# B&R Automation Studio project RTFProj (part 5)

##### test.c
```c
/*********************************************************************************************
* B&R Automation - Perfection in Automation (https://www.br-automation.com)
    ******************************************************************************************
    * Program 	    : Master's Thesis - Soccer Table (Table Football - real game)
    * Author  	    : Roman Parak
    * Created 	    : date ...
	* University    : Brno University of Technology(BUT)
	* Faculty       : Faculty of Mechanical Engineering(FME)
	* Study Program : Applied Computer Science and Control
	* Institute     : Institute of Automation and Computer Science
**********************************************************************************************
* Implementation OF PROGRAM Test(Real_Game/Technology/Test/Program/test.h)
**********************************************************************************************/

/*************************** LIBRARIES *********************************/
#include <bur/plc.h>
#include <bur/plctypes.h>
#include <stdio.h>
#include <math.h>

#include "rp_funcx1.h"
#include "Structures/test_str.h"
#include "Functions/test_fce.h"

#ifdef _DEFAULT_INCLUDES
	#include <AsDefault.h>
#endif

/*************************** DEFINITIONS *******************************/
#define EACH_FORMATION 1;

/************************ LOCAL VARIABLES ******************************/
// struct - MpAlarmX
_LOCAL MpAlarmXListUIConnectType AlarmListUI_ConnectType;
_LOCAL MpAlarmXHistoryUIConnectType AlarmHistoryUI_ConnectType;
// udint
_LOCAL UDINT alarm_device_address;
// bool
_LOCAL BOOL start;
_LOCAL BOOL stop;
// usint
_LOCAL USINT max_numberOfFormation;
_LOCAL USINT i_axisNum;
// lreal
_LOCAL LREAL temp_lin;
_LOCAL LREAL temp_rot;
_LOCAL LREAL define_posRotary;
_LOCAL LREAL angle_ofRotation;
// state machine
_LOCAL rp_MainSteps soccer_step;

/**********************************************************************************************************/
/********************************************** INIT PROGRAM **********************************************/
/**********************************************************************************************************/
void _INIT ProgramInit(void)
{
    /*********************************** Declaration variables **********************************/
    // generally
    max_numberOfFormation = EACH_FORMATION;

    // axis type -> MAPP
    // linear
    gLinkAxes_linear[0] = gk_mappAxisL;
    /*
    gLinkAxes_linear[1] = df_mappAxisL;
    gLinkAxes_linear[2] = md_mappAxisL;
    gLinkAxes_linear[3] = fw_mappAxisL;
    */
    // rotary
    gLinkAxes_rotary[0] = gk_mappAxisR;
   	/*
    gLinkAxes_rotary[1] = df_mappAxisR;
    gLinkAxes_rotary[2] = md_mappAxisR;
    gLinkAxes_rotary[3] = fw_mappAxisR;
    */
    /************************************ Control of AlarmX ************************************/

    // adjustment device name
    alarm_device_address = (UDINT) strcpy(mp_alarmX.deviceName_no1_exp,"EXPORT_HISTORY");
    // MpAlarmX Core
    mp_alarmX.mp_core.MpLink         = &gAlarmXCore;
    mp_alarmX.mp_core.Enable         = 1;
    // MpAlarmX ListUI
    mp_alarmX.mp_listUI.MpLink       = &gAlarmXCore;
    mp_alarmX.mp_listUI.Enable       = 1;
    mp_alarmX.mp_listUI.UIConnect    = &AlarmListUI_ConnectType;
    // MpAlarmX History
    mp_alarmX.mp_history.MpLink      = &gAlarmXHistory;
    mp_alarmX.mp_history.Enable      = 1;
    mp_alarmX.mp_history.DeviceName  = &mp_alarmX.deviceName_no1_exp;
    // MpAlarmX HistoryUI
    mp_alarmX.mp_historyUI.MpLink    = &gAlarmXHistory;
    mp_alarmX.mp_historyUI.Enable    = 1;
    mp_alarmX.mp_historyUI.UIConnect = &AlarmHistoryUI_ConnectType;

    /************************************* Control of Axes **************************************/

    for(i_axisNum = 0; i_axisNum <= max_numberOfFormation - 1; i_axisNum++){
        // initialization ACOPOS variables through function(get_axisParam), that returns two variables type of UDINT
        // into the structure -> axesAcopos(have two parameters : linear, rotary)
        axis_acopos = get_axisParam(i_axisNum);
        // linear -> LinMot
        // linear axis basic
        mp_Axis.mp_axisLinear[i_axisNum].Enable     = 1;
        mp_Axis.mp_axisLinear[i_axisNum].MpLink     = &gLinkAxes_linear[i_axisNum];
        mp_Axis.mp_axisLinear[i_axisNum].Parameters = &mp_Axis.param_axisLinear[i_axisNum];
        mp_Axis.mp_axisLinear[i_axisNum].Axis       = axis_acopos.linear;
		// initialization parameters -> linear
		mp_Axis.param_axisLinear[i_axisNum].Home.Mode 	 		 	     = mpAXIS_HOME_MODE_BLOCK_TORQUE;
		mp_Axis.param_axisLinear[i_axisNum].Home.Position 		  	     = 900;
		mp_Axis.param_axisLinear[i_axisNum].Home.StartVelocity   		 = 350;
		mp_Axis.param_axisLinear[i_axisNum].Home.HomingVelocity  		 = 450;
		mp_Axis.param_axisLinear[i_axisNum].Home.Acceleration    		 = 350;
		mp_Axis.param_axisLinear[i_axisNum].Home.StartDirection  		 = mpAXIS_HOME_DIR_POSITIVE;
		mp_Axis.param_axisLinear[i_axisNum].Home.HomingDirection 		 = mpAXIS_HOME_DIR_NEGATIVE;
		mp_Axis.param_axisLinear[i_axisNum].Home.TorqueLimit	 		 = 0.05;
		mp_Axis.param_axisLinear[i_axisNum].Home.PositionErrorStopLimit	 = 900;
        // linear cyclic set
        mp_Axis.mp_cyclicSetLinear[i_axisNum].Enable     = 1;
        mp_Axis.mp_cyclicSetLinear[i_axisNum].MpLink     = &gLinkAxes_linear[i_axisNum];
        mp_Axis.mp_cyclicSetLinear[i_axisNum].Parameters = &mp_Axis.param_cyclicSetLinear[i_axisNum];
		// config
		mp_Axis.mp_configAxisLinear[i_axisNum].Enable 		 = 1;
		mp_Axis.mp_configAxisLinear[i_axisNum].MpLink 		 = &gLinkAxes_linear[i_axisNum];
		mp_Axis.mp_configAxisLinear[i_axisNum].Configuration = &mp_Axis.param_configAxisLinear[i_axisNum];
        // rotary -> EnDat
        // rotary axis basic
        mp_Axis.mp_axisRotary[i_axisNum].Enable     = 1;
        mp_Axis.mp_axisRotary[i_axisNum].MpLink     = &gLinkAxes_rotary[i_axisNum];
        mp_Axis.mp_axisRotary[i_axisNum].Parameters = &mp_Axis.param_axisRotary[i_axisNum];
        mp_Axis.mp_axisRotary[i_axisNum].Axis       = axis_acopos.rotary;
        // rotary cyclic set
        mp_Axis.mp_cyclicSetRotary[i_axisNum].Enable     = 1;
        mp_Axis.mp_cyclicSetRotary[i_axisNum].MpLink     = &gLinkAxes_rotary[i_axisNum];
        mp_Axis.mp_cyclicSetRotary[i_axisNum].Parameters = &mp_Axis.param_cyclicSetRotary[i_axisNum];
		// config
		mp_Axis.mp_configAxisRotary[i_axisNum].Enable 		 = 1;
		mp_Axis.mp_configAxisRotary[i_axisNum].MpLink 		 = &gLinkAxes_rotary[i_axisNum];
		mp_Axis.mp_configAxisRotary[i_axisNum].Configuration = &mp_Axis.param_configAxisRotary[i_axisNum];
		// temperature - linear
		mp_Axis.param_axisLinear[i_axisNum].CyclicRead.MotorTempMode = mpAXIS_READ_POLLING_1s;
		// temperature - rotary
		mp_Axis.param_axisRotary[i_axisNum].CyclicRead.MotorTempMode = mpAXIS_READ_POLLING_1s;
    }
	// initializatiom temp
	temp_lin = 0;
	temp_rot = 0;
	define_posRotary = 118520697;
	angle_ofRotation = 0;
	// initialization state machine
	soccer_step = STEP_INITIALIZATION;
}

/**********************************************************************************************************/
/********************************************** MAIN PROGRAM **********************************************/
/**********************************************************************************************************/
void _CYCLIC ProgramCyclic(void)
{
	// initializatiom temp
	temp_lin = mp_Axis.mp_axisLinear[0].Info.CyclicRead.MotorTemperature.Value;
	temp_rot = mp_Axis.mp_axisRotary[0].Info.CyclicRead.MotorTemperature.Value;

	switch(soccer_step)
	{
		case STEP_INITIALIZATION:
			{
				if(mp_Axis.mp_axisLinear[0].Active == 1 && mp_Axis.mp_axisRotary[0].Active == 1){
					angle_ofRotation = get_rotationalPostition(mp_Axis.mp_axisRotary[0].Position,define_posRotary);

					if(labs(angle_ofRotation) <= 3600){
						mp_Axis.param_axisRotary[0].Home.Position = angle_ofRotation;
						soccer_step = STEP_INITIALIZATION0;
					}
				}
			}
			break;
		case STEP_INITIALIZATION0:
			{
				if(mp_Axis.mp_axisLinear[0].Error == 1 && mp_Axis.mp_axisRotary[0].Error == 0){
					soccer_step = STEP_ERROR1;
				}else if(mp_Axis.mp_axisLinear[0].StatusID < 0 || mp_Axis.mp_axisRotary[0].StatusID < 0){
					soccer_step = STEP_ERROR2;
				}else {
					if(mp_Axis.mp_axisLinear[0].IsHomed == 1 && mp_Axis.mp_axisRotary[0].IsHomed == 1){
						soccer_step = STEP_RUN7;
					}else{
						soccer_step = STEP_INITIALIZATION1;
					}
				}
			}
			break;
		case STEP_INITIALIZATION1:
			{
				if(start == 1){
					mp_Axis.mp_axisLinear[0].Power = 1;
					mp_Axis.mp_axisRotary[0].Power = 1;

					if(mp_alarmX.mp_core.ActiveAlarms == 1){
						soccer_step = STEP_ERROR1;
					}else if(stop == 1){
						soccer_step = STEP_STOP1;
					}else{
						if(mp_Axis.mp_axisLinear[0].PowerOn == 1 && mp_Axis.mp_axisRotary[0].PowerOn == 1){
							soccer_step = STEP_INITIALIZATION2;
						}
					}
				}
			}
			break;
		case STEP_INITIALIZATION2:
			{
				mp_Axis.mp_axisLinear[0].Update = 1;
				mp_Axis.mp_axisRotary[0].Update = 1;

				if(mp_alarmX.mp_core.ActiveAlarms == 1){
					soccer_step = STEP_ERROR1;
				}else if(stop == 1){
					soccer_step = STEP_STOP1;
				}else{
					if(mp_Axis.mp_axisLinear[0].UpdateDone == 1 && mp_Axis.mp_axisRotary[0].UpdateDone == 1){
						mp_Axis.mp_axisLinear[0].Update = 0;
						mp_Axis.mp_axisRotary[0].Update = 0;
						soccer_step = STEP_INITIALIZATION3;
					}
				}
			}
			break;
		case STEP_INITIALIZATION3:
			{
				mp_Axis.mp_axisRotary[0].Home = 1;

				if(mp_alarmX.mp_core.ActiveAlarms == 1){
					soccer_step = STEP_ERROR1;
				}else if(stop == 1){
					soccer_step = STEP_STOP1;
				}else{
					if(mp_Axis.mp_axisRotary[0].IsHomed == 1){
						mp_Axis.mp_axisRotary[0].Home = 0;
						soccer_step = STEP_INITIALIZATION4;
					}
				}
			}
			break;
		case STEP_INITIALIZATION4:
			{
				mp_Axis.param_cyclicSetRotary[0].Acceleration = 2000;
				mp_Axis.param_cyclicSetRotary[0].Deceleration = 2000;
				mp_Axis.param_cyclicSetRotary[0].PositionModeMaxVelocity = 85000;
				mp_Axis.mp_cyclicSetRotary[0].Velocity 	 = 1000;
				mp_Axis.mp_cyclicSetRotary[0].Position	 = 0;

				mp_Axis.mp_cyclicSetRotary[0].Update = 1;
				if(mp_alarmX.mp_core.ActiveAlarms == 1){
					soccer_step = STEP_ERROR1;
				}else if(stop == 1){
					soccer_step = STEP_STOP1;
				}else{
					if(mp_Axis.mp_cyclicSetRotary[0].UpdateDone == 1){
						mp_Axis.mp_cyclicSetRotary[0].Update = 0;
						if(mp_Axis.mp_cyclicSetRotary[0].CommandBusy == 0 && mp_Axis.mp_cyclicSetRotary[0].CyclicSetActive == 0){
							soccer_step = STEP_INITIALIZATION5;
						}
					}
				}
			}
			break;
		case STEP_INITIALIZATION5:
			{
				mp_Axis.mp_cyclicSetRotary[0].CyclicPosition = 1;
				if(mp_alarmX.mp_core.ActiveAlarms == 1){
					soccer_step = STEP_ERROR1;
				}else if(stop == 1){
					soccer_step = STEP_STOP1;
				}else{
					if(mp_Axis.mp_cyclicSetRotary[0].Info.SlavePosition == 0){
						mp_Axis.mp_cyclicSetRotary[0].CyclicPosition = 0;
						if(mp_Axis.mp_cyclicSetRotary[0].CommandBusy == 0 && mp_Axis.mp_cyclicSetRotary[0].CyclicSetActive == 0){
							soccer_step = STEP_INITIALIZATION6;
						}
					}
				}
			}
			break;
		case STEP_INITIALIZATION6:
			{
				mp_Axis.mp_axisLinear[0].Home = 1;

				if(mp_alarmX.mp_core.ActiveAlarms == 1){
					soccer_step = STEP_ERROR1;
				}else if(stop == 1){
					soccer_step = STEP_STOP1;
				}else{
					if(mp_Axis.mp_axisLinear[0].IsHomed == 1){
						mp_Axis.mp_axisLinear[0].Home = 0;
						soccer_step = STEP_START;
					}
				}
			}
			break;
		case STEP_START:
			{
				mp_Axis.param_cyclicSetLinear[0].Acceleration = 400000;
				mp_Axis.param_cyclicSetLinear[0].Deceleration = 400000;
				mp_Axis.param_cyclicSetLinear[0].PositionModeMaxVelocity = 30000;
				mp_Axis.mp_cyclicSetLinear[0].Velocity = 19000;
				mp_Axis.mp_cyclicSetLinear[0].Position = 0;

				mp_Axis.mp_cyclicSetLinear[0].Update = 1;
				if(mp_alarmX.mp_core.ActiveAlarms == 1){
					soccer_step = STEP_ERROR1;
				}else if(stop == 1){
					soccer_step = STEP_STOP1;
				}else{
					if(mp_Axis.mp_cyclicSetLinear[0].UpdateDone == 1){
						mp_Axis.mp_cyclicSetLinear[0].Update = 0;
						if(mp_Axis.mp_cyclicSetLinear[0].CommandBusy == 0 && mp_Axis.mp_cyclicSetLinear[0].CyclicSetActive == 0){
							soccer_step = STEP_RUN1;
						}
					}
				}
			}
			break;
		case STEP_RUN1:
			{
				mp_Axis.mp_cyclicSetLinear[0].CyclicPosition = 1;
				if(mp_alarmX.mp_core.ActiveAlarms == 1){
					soccer_step = STEP_ERROR1;
				}else if(stop == 1){
					soccer_step = STEP_STOP1;
				}else{
					if(mp_Axis.mp_cyclicSetLinear[0].Info.SlavePosition == 0){
						mp_Axis.mp_cyclicSetLinear[0].CyclicPosition = 0;
						if(mp_Axis.mp_cyclicSetLinear[0].CommandBusy == 0 && mp_Axis.mp_cyclicSetLinear[0].CyclicSetActive == 0){
							soccer_step = STEP_RUN2;
						}
					}
				}
			}
			break;
		case STEP_RUN2:
			{
				mp_Axis.param_cyclicSetRotary[0].Acceleration = 125000;
				mp_Axis.param_cyclicSetRotary[0].Deceleration = 125000;
				mp_Axis.param_cyclicSetRotary[0].PositionModeMaxVelocity = 85000;
				mp_Axis.mp_cyclicSetRotary[0].Velocity 	 = 10000;
				mp_Axis.mp_cyclicSetRotary[0].Position	 = -800;

				mp_Axis.mp_cyclicSetRotary[0].Update = 1;
				if(mp_alarmX.mp_core.ActiveAlarms == 1){
					soccer_step = STEP_ERROR1;
				}else if(stop == 1){
					soccer_step = STEP_STOP1;
				}else{
					if(mp_Axis.mp_cyclicSetRotary[0].UpdateDone == 1){
						mp_Axis.mp_cyclicSetRotary[0].Update = 0;
						if(mp_Axis.mp_cyclicSetRotary[0].CommandBusy == 0 && mp_Axis.mp_cyclicSetRotary[0].CyclicSetActive == 0){
							soccer_step = STEP_RUN3;
						}
					}
				}
			}
			break;
		case STEP_RUN3:
			{
				mp_Axis.mp_cyclicSetRotary[0].CyclicPosition = 1;
				if(mp_alarmX.mp_core.ActiveAlarms == 1){
					soccer_step = STEP_ERROR1;
				}else if(stop == 1){
					soccer_step = STEP_STOP1;
				}else{
					if(mp_Axis.mp_cyclicSetRotary[0].Info.SlavePosition == -800){
						mp_Axis.mp_cyclicSetRotary[0].CyclicPosition = 0;
						if(mp_Axis.mp_cyclicSetRotary[0].CommandBusy == 0 && mp_Axis.mp_cyclicSetRotary[0].CyclicSetActive == 0){
							soccer_step = STEP_RUN4;
						}
					}
				}
			}
			break;
		case STEP_RUN4:
			{
				mp_Axis.param_cyclicSetRotary[0].Acceleration = 125000;
				mp_Axis.param_cyclicSetRotary[0].Deceleration = 125000;
				mp_Axis.param_cyclicSetRotary[0].PositionModeMaxVelocity = 85000;
				mp_Axis.mp_cyclicSetRotary[0].Velocity 	 = 10000;
				mp_Axis.mp_cyclicSetRotary[0].Position	 = 800;

				mp_Axis.mp_cyclicSetRotary[0].Update = 1;
				if(mp_alarmX.mp_core.ActiveAlarms == 1){
					soccer_step = STEP_ERROR1;
				}else if(stop == 1){
					soccer_step = STEP_STOP1;
				}else{
					if(mp_Axis.mp_cyclicSetRotary[0].UpdateDone == 1){
						mp_Axis.mp_cyclicSetRotary[0].Update = 0;
						if(mp_Axis.mp_cyclicSetRotary[0].CommandBusy == 0 && mp_Axis.mp_cyclicSetRotary[0].CyclicSetActive == 0){
							soccer_step = STEP_RUN5;
						}
					}
				}
			}
			break;
		case STEP_RUN5:
			{
				mp_Axis.mp_cyclicSetRotary[0].CyclicPosition = 1;
				if(mp_alarmX.mp_core.ActiveAlarms == 1){
					soccer_step = STEP_ERROR1;
				}else if(stop == 1){
					soccer_step = STEP_STOP1;
				}else{
					if(mp_Axis.mp_cyclicSetRotary[0].Info.SlavePosition == 800){
						mp_Axis.mp_cyclicSetRotary[0].CyclicPosition = 0;
						if(mp_Axis.mp_cyclicSetRotary[0].CommandBusy == 0 && mp_Axis.mp_cyclicSetRotary[0].CyclicSetActive == 0){
							soccer_step = STEP_RUN6;
						}
					}
				}
			}
			break;
		case STEP_RUN6:
			{
				/*======================= END HOME =======================*/
				mp_Axis.param_cyclicSetRotary[0].Acceleration = 125000;
				mp_Axis.param_cyclicSetRotary[0].Deceleration = 125000;
				mp_Axis.param_cyclicSetRotary[0].PositionModeMaxVelocity = 85000;
				mp_Axis.mp_cyclicSetRotary[0].Velocity 	 = 10000;
				mp_Axis.mp_cyclicSetRotary[0].Position	 = 0;

				mp_Axis.mp_cyclicSetRotary[0].Update = 1;
				if(mp_alarmX.mp_core.ActiveAlarms == 1){
					soccer_step = STEP_ERROR1;
				}else if(stop == 1){
					soccer_step = STEP_STOP1;
				}else{
					if(mp_Axis.mp_cyclicSetRotary[0].UpdateDone == 1){
						mp_Axis.mp_cyclicSetRotary[0].Update = 0;
						if(mp_Axis.mp_cyclicSetRotary[0].CommandBusy == 0 && mp_Axis.mp_cyclicSetRotary[0].CyclicSetActive == 0){
							soccer_step = STEP_RUN7;
						}
					}
				}
			}
			break;
		case STEP_RUN7:
			{
				/*======================= START CYCLE =======================*/
				mp_Axis.mp_cyclicSetRotary[0].CyclicPosition = 1;
				if(mp_alarmX.mp_core.ActiveAlarms == 1){
					soccer_step = STEP_ERROR1;
				}else if(stop == 1){
					soccer_step = STEP_STOP1;
				}else{
					if(mp_Axis.mp_cyclicSetRotary[0].Info.SlavePosition == 0){
						mp_Axis.mp_cyclicSetRotary[0].CyclicPosition = 0;
						if(mp_Axis.mp_cyclicSetRotary[0].CommandBusy == 0 && mp_Axis.mp_cyclicSetRotary[0].CyclicSetActive == 0){
							soccer_step = STEP_RUN8;
						}
					}
				}
			}
			break;
		case STEP_RUN8:
			{
				// 250000,20000
				mp_Axis.param_cyclicSetLinear[0].Acceleration = 125000;
				mp_Axis.param_cyclicSetLinear[0].Deceleration = 125000;
				mp_Axis.param_cyclicSetLinear[0].PositionModeMaxVelocity = 30000;
				mp_Axis.mp_cyclicSetLinear[0].Velocity = 10000;
				mp_Axis.mp_cyclicSetLinear[0].Position = -800;

				mp_Axis.mp_cyclicSetLinear[0].Update = 1;
				if(mp_alarmX.mp_core.ActiveAlarms == 1){
					soccer_step = STEP_ERROR1;
				}else if(stop == 1){
					soccer_step = STEP_STOP1;
				}else{
					if(mp_Axis.mp_cyclicSetLinear[0].UpdateDone == 1){
						mp_Axis.mp_cyclicSetLinear[0].Update = 0;
						if(mp_Axis.mp_cyclicSetLinear[0].CommandBusy == 0 && mp_Axis.mp_cyclicSetLinear[0].CyclicSetActive == 0){
							soccer_step = STEP_RUN9;
						}
					}
				}
			}
			break;
		case STEP_RUN9:
			{
				mp_Axis.mp_cyclicSetLinear[0].CyclicPosition = 1;
				if(mp_alarmX.mp_core.ActiveAlarms == 1){
					soccer_step = STEP_ERROR1;
				}else if(stop == 1){
					soccer_step = STEP_STOP1;
				}else{
					if(mp_Axis.mp_cyclicSetLinear[0].Info.SlavePosition == -800){
						mp_Axis.mp_cyclicSetLinear[0].CyclicPosition = 0;
						if(mp_Axis.mp_cyclicSetLinear[0].CommandBusy == 0 && mp_Axis.mp_cyclicSetLinear[0].CyclicSetActive == 0){
							soccer_step = STEP_RUN10; // STEP_RUN24
						}
					}
				}
			}
			break;
		case STEP_RUN10:
			{
				mp_Axis.param_cyclicSetRotary[0].Acceleration = 31250;
				mp_Axis.param_cyclicSetRotary[0].Deceleration = 31250;
				mp_Axis.param_cyclicSetRotary[0].PositionModeMaxVelocity = 85000;
				mp_Axis.mp_cyclicSetRotary[0].Velocity 	 = 5000;
				mp_Axis.mp_cyclicSetRotary[0].Position	 = -800;

				mp_Axis.mp_cyclicSetRotary[0].Update = 1;
				if(mp_alarmX.mp_core.ActiveAlarms == 1){
					soccer_step = STEP_ERROR1;
				}else if(stop == 1){
					soccer_step = STEP_STOP1;
				}else{
					if(mp_Axis.mp_cyclicSetRotary[0].UpdateDone == 1){
						mp_Axis.mp_cyclicSetRotary[0].Update = 0;
						if(mp_Axis.mp_cyclicSetRotary[0].CommandBusy == 0 && mp_Axis.mp_cyclicSetRotary[0].CyclicSetActive == 0){
							soccer_step = STEP_RUN11;
						}
					}
				}
			}
			break;
		case STEP_RUN11:
			{
				mp_Axis.mp_cyclicSetRotary[0].CyclicPosition = 1;
				if(mp_alarmX.mp_core.ActiveAlarms == 1){
					soccer_step = STEP_ERROR1;
				}else if(stop == 1){
					soccer_step = STEP_STOP1;
				}else{
					if(mp_Axis.mp_cyclicSetRotary[0].Info.SlavePosition == -800){
						mp_Axis.mp_cyclicSetRotary[0].CyclicPosition = 0;
						if(mp_Axis.mp_cyclicSetRotary[0].CommandBusy == 0 && mp_Axis.mp_cyclicSetRotary[0].CyclicSetActive == 0){
							soccer_step = STEP_RUN12;
						}
					}
				}
			}
			break;
		case STEP_RUN12:
			{
				mp_Axis.param_cyclicSetRotary[0].Acceleration = 31250;
				mp_Axis.param_cyclicSetRotary[0].Deceleration = 31250;
				mp_Axis.param_cyclicSetRotary[0].PositionModeMaxVelocity = 85000;
				mp_Axis.mp_cyclicSetRotary[0].Velocity 	 = 5000;
				mp_Axis.mp_cyclicSetRotary[0].Position	 = 800;

				mp_Axis.mp_cyclicSetRotary[0].Update = 1;
				if(mp_alarmX.mp_core.ActiveAlarms == 1){
					soccer_step = STEP_ERROR1;
				}else if(stop == 1){
					soccer_step = STEP_STOP1;
				}else{
					if(mp_Axis.mp_cyclicSetRotary[0].UpdateDone == 1){
						mp_Axis.mp_cyclicSetRotary[0].Update = 0;
						if(mp_Axis.mp_cyclicSetRotary[0].CommandBusy == 0 && mp_Axis.mp_cyclicSetRotary[0].CyclicSetActive == 0){
							soccer_step = STEP_RUN13;
						}
					}
				}
			}
			break;
		case STEP_RUN13:
			{
				mp_Axis.mp_cyclicSetRotary[0].CyclicPosition = 1;
				if(mp_alarmX.mp_core.ActiveAlarms == 1){
					soccer_step = STEP_ERROR1;
				}else if(stop == 1){
					soccer_step = STEP_STOP1;
				}else{
					if(mp_Axis.mp_cyclicSetRotary[0].Info.SlavePosition == 800){
						mp_Axis.mp_cyclicSetRotary[0].CyclicPosition = 0;
						if(mp_Axis.mp_cyclicSetRotary[0].CommandBusy == 0 && mp_Axis.mp_cyclicSetRotary[0].CyclicSetActive == 0){
							soccer_step = STEP_RUN14;
						}
					}
				}
			}
			break;
		case STEP_RUN14:
			{
				mp_Axis.param_cyclicSetRotary[0].Acceleration = 31250;
				mp_Axis.param_cyclicSetRotary[0].Deceleration = 31250;
				mp_Axis.param_cyclicSetRotary[0].PositionModeMaxVelocity = 85000;
				mp_Axis.mp_cyclicSetRotary[0].Velocity 	 = 5000;
				mp_Axis.mp_cyclicSetRotary[0].Position	 = 0;

				mp_Axis.mp_cyclicSetRotary[0].Update = 1;
				if(mp_alarmX.mp_core.ActiveAlarms == 1){
					soccer_step = STEP_ERROR1;
				}else if(stop == 1){
					soccer_step = STEP_STOP1;
				}else{
					if(mp_Axis.mp_cyclicSetRotary[0].UpdateDone == 1){
						mp_Axis.mp_cyclicSetRotary[0].Update = 0;
						if(mp_Axis.mp_cyclicSetRotary[0].CommandBusy == 0 && mp_Axis.mp_cyclicSetRotary[0].CyclicSetActive == 0){
							soccer_step = STEP_RUN15;
						}
					}
				}
			}
			break;
		case STEP_RUN15:
			{
				mp_Axis.mp_cyclicSetRotary[0].CyclicPosition = 1;
				if(mp_alarmX.mp_core.ActiveAlarms == 1){
					soccer_step = STEP_ERROR1;
				}else if(stop == 1){
					soccer_step = STEP_STOP1;
				}else{
					if(mp_Axis.mp_cyclicSetRotary[0].Info.SlavePosition == 0){
						mp_Axis.mp_cyclicSetRotary[0].CyclicPosition = 0;
						if(mp_Axis.mp_cyclicSetRotary[0].CommandBusy == 0 && mp_Axis.mp_cyclicSetRotary[0].CyclicSetActive == 0){
							soccer_step = STEP_RUN16; // STEP_RUN24
						}
					}
				}
			}
			break;
		case STEP_RUN16:
			{
				mp_Axis.param_cyclicSetLinear[0].Acceleration = 600;
				mp_Axis.param_cyclicSetLinear[0].Deceleration = 600;
				mp_Axis.param_cyclicSetLinear[0].PositionModeMaxVelocity = 30000;
				mp_Axis.mp_cyclicSetLinear[0].Velocity = 2500;
				mp_Axis.mp_cyclicSetLinear[0].Position = 0;

				mp_Axis.mp_cyclicSetLinear[0].Update = 1;
				if(mp_alarmX.mp_core.ActiveAlarms == 1){
					soccer_step = STEP_ERROR1;
				}else if(stop == 1){
					soccer_step = STEP_STOP1;
				}else{
					if(mp_Axis.mp_cyclicSetLinear[0].UpdateDone == 1){
						mp_Axis.mp_cyclicSetLinear[0].Update = 0;
						if(mp_Axis.mp_cyclicSetLinear[0].CommandBusy == 0 && mp_Axis.mp_cyclicSetLinear[0].CyclicSetActive == 0){
							soccer_step = STEP_RUN17;
						}
					}
				}
			}
			break;
		case STEP_RUN17:
			{
				mp_Axis.mp_cyclicSetLinear[0].CyclicPosition = 1;
				if(mp_alarmX.mp_core.ActiveAlarms == 1){
					soccer_step = STEP_ERROR1;
				}else if(stop == 1){
					soccer_step = STEP_STOP1;
				}else{
					if(mp_Axis.mp_cyclicSetLinear[0].Info.SlavePosition == 0){
						mp_Axis.mp_cyclicSetLinear[0].CyclicPosition = 0;
						if(mp_Axis.mp_cyclicSetLinear[0].CommandBusy == 0 && mp_Axis.mp_cyclicSetLinear[0].CyclicSetActive == 0){
							soccer_step = STEP_RUN18;
						}
					}
				}
			}
			break;
		case STEP_RUN18:
			{
				mp_Axis.param_cyclicSetRotary[0].Acceleration = 3900000;
				mp_Axis.param_cyclicSetRotary[0].Deceleration = 3900000;
				mp_Axis.param_cyclicSetRotary[0].PositionModeMaxVelocity = 85000;
				mp_Axis.mp_cyclicSetRotary[0].Velocity 	 = 84000;
				mp_Axis.mp_cyclicSetRotary[0].Position	 = -800;

				mp_Axis.mp_cyclicSetRotary[0].Update = 1;
				if(mp_alarmX.mp_core.ActiveAlarms == 1){
					soccer_step = STEP_ERROR1;
				}else if(stop == 1){
					soccer_step = STEP_STOP1;
				}else{
					if(mp_Axis.mp_cyclicSetRotary[0].UpdateDone == 1){
						mp_Axis.mp_cyclicSetRotary[0].Update = 0;
						if(mp_Axis.mp_cyclicSetRotary[0].CommandBusy == 0 && mp_Axis.mp_cyclicSetRotary[0].CyclicSetActive == 0){
							soccer_step = STEP_RUN19;
						}
					}
				}
			}
			break;
		case STEP_RUN19:
			{
				mp_Axis.mp_cyclicSetRotary[0].CyclicPosition = 1;
				if(mp_alarmX.mp_core.ActiveAlarms == 1){
					soccer_step = STEP_ERROR1;
				}else if(stop == 1){
					soccer_step = STEP_STOP1;
				}else{
					if(mp_Axis.mp_cyclicSetRotary[0].Info.SlavePosition == -800){
						mp_Axis.mp_cyclicSetRotary[0].CyclicPosition = 0;
						if(mp_Axis.mp_cyclicSetRotary[0].CommandBusy == 0 && mp_Axis.mp_cyclicSetRotary[0].CyclicSetActive == 0){
							soccer_step = STEP_RUN20;
						}
					}
				}
			}
			break;
		case STEP_RUN20:
			{
				mp_Axis.param_cyclicSetRotary[0].Acceleration = 3900000;
				mp_Axis.param_cyclicSetRotary[0].Deceleration = 3900000;
				mp_Axis.param_cyclicSetRotary[0].PositionModeMaxVelocity = 85000;
				mp_Axis.mp_cyclicSetRotary[0].Velocity 	 = 80000;
				mp_Axis.mp_cyclicSetRotary[0].Position	 = 800;

				mp_Axis.mp_cyclicSetRotary[0].Update = 1;
				if(mp_alarmX.mp_core.ActiveAlarms == 1){
					soccer_step = STEP_ERROR1;
				}else if(stop == 1){
					soccer_step = STEP_STOP1;
				}else{
					if(mp_Axis.mp_cyclicSetRotary[0].UpdateDone == 1){
						mp_Axis.mp_cyclicSetRotary[0].Update = 0;
						if(mp_Axis.mp_cyclicSetRotary[0].CommandBusy == 0 && mp_Axis.mp_cyclicSetRotary[0].CyclicSetActive == 0){
							soccer_step = STEP_RUN21;
						}
					}
				}
			}
			break;
		case STEP_RUN21:
			{
				mp_Axis.mp_cyclicSetRotary[0].CyclicPosition = 1;
				if(mp_alarmX.mp_core.ActiveAlarms == 1){
					soccer_step = STEP_ERROR1;
				}else if(stop == 1){
					soccer_step = STEP_STOP1;
				}else{
					if(mp_Axis.mp_cyclicSetRotary[0].Info.SlavePosition == 800){
						mp_Axis.mp_cyclicSetRotary[0].CyclicPosition = 0;
						if(mp_Axis.mp_cyclicSetRotary[0].CommandBusy == 0 && mp_Axis.mp_cyclicSetRotary[0].CyclicSetActive == 0){
							soccer_step = STEP_RUN22;
						}
					}
				}
			}
			break;
		case STEP_RUN22:
			{
				mp_Axis.param_cyclicSetRotary[0].Acceleration = 3900000;
				mp_Axis.param_cyclicSetRotary[0].Deceleration = 3900000;
				mp_Axis.param_cyclicSetRotary[0].PositionModeMaxVelocity = 85000;
				mp_Axis.mp_cyclicSetRotary[0].Velocity 	 = 80000;
				mp_Axis.mp_cyclicSetRotary[0].Position	 = 0;

				mp_Axis.mp_cyclicSetRotary[0].Update = 1;
				if(mp_alarmX.mp_core.ActiveAlarms == 1){
					soccer_step = STEP_ERROR1;
				}else if(stop == 1){
					soccer_step = STEP_STOP1;
				}else{
					if(mp_Axis.mp_cyclicSetRotary[0].UpdateDone == 1){
						mp_Axis.mp_cyclicSetRotary[0].Update = 0;
						if(mp_Axis.mp_cyclicSetRotary[0].CommandBusy == 0 && mp_Axis.mp_cyclicSetRotary[0].CyclicSetActive == 0){
							soccer_step = STEP_RUN23;
						}
					}
				}
			}
			break;
		case STEP_RUN23:
			{
				mp_Axis.mp_cyclicSetRotary[0].CyclicPosition = 1;
				if(mp_alarmX.mp_core.ActiveAlarms == 1){
					soccer_step = STEP_ERROR1;
				}else if(stop == 1){
					soccer_step = STEP_STOP1;
				}else{
					if(mp_Axis.mp_cyclicSetRotary[0].Info.SlavePosition == 0){
						mp_Axis.mp_cyclicSetRotary[0].CyclicPosition = 0;
						if(mp_Axis.mp_cyclicSetRotary[0].CommandBusy == 0 && mp_Axis.mp_cyclicSetRotary[0].CyclicSetActive == 0){
							soccer_step = STEP_RUN24;
						}
					}
				}
			}
			break;
		case STEP_RUN24:
			{
				// 250000, 20000
				mp_Axis.param_cyclicSetLinear[0].Acceleration = 281250;
				mp_Axis.param_cyclicSetLinear[0].Deceleration = 281250;
				mp_Axis.param_cyclicSetLinear[0].PositionModeMaxVelocity = 30000;
				mp_Axis.mp_cyclicSetLinear[0].Velocity = 15000;
				mp_Axis.mp_cyclicSetLinear[0].Position = 800;

				mp_Axis.mp_cyclicSetLinear[0].Update = 1;
				if(mp_alarmX.mp_core.ActiveAlarms == 1){
					soccer_step = STEP_ERROR1;
				}else if(stop == 1){
					soccer_step = STEP_STOP1;
				}else{
					if(mp_Axis.mp_cyclicSetLinear[0].UpdateDone == 1){
						mp_Axis.mp_cyclicSetLinear[0].Update = 0;
						if(mp_Axis.mp_cyclicSetLinear[0].CommandBusy == 0 && mp_Axis.mp_cyclicSetLinear[0].CyclicSetActive == 0){
							soccer_step = STEP_RUN25;
						}
					}
				}
			}
			break;
		case STEP_RUN25:
			{
				mp_Axis.mp_cyclicSetLinear[0].CyclicPosition = 1;
				if(mp_alarmX.mp_core.ActiveAlarms == 1){
					soccer_step = STEP_ERROR1;
				}else if(stop == 1){
					soccer_step = STEP_STOP1;
				}else{
					if(mp_Axis.mp_cyclicSetLinear[0].Info.SlavePosition == 800){
						mp_Axis.mp_cyclicSetLinear[0].CyclicPosition = 0;
						if(mp_Axis.mp_cyclicSetLinear[0].CommandBusy == 0 && mp_Axis.mp_cyclicSetLinear[0].CyclicSetActive == 0){
							soccer_step = STEP_RUN26; // STEP_RUN8
						}
					}
				}
			}
			break;
		case STEP_RUN26:
			{
				mp_Axis.param_cyclicSetRotary[0].Acceleration = 3125000;
				mp_Axis.param_cyclicSetRotary[0].Deceleration = 3125000;
				mp_Axis.param_cyclicSetRotary[0].PositionModeMaxVelocity = 85000;
				mp_Axis.mp_cyclicSetRotary[0].Velocity 	 = 50000;
				mp_Axis.mp_cyclicSetRotary[0].Position	 = -800;

				mp_Axis.mp_cyclicSetRotary[0].Update = 1;
				if(mp_alarmX.mp_core.ActiveAlarms == 1){
					soccer_step = STEP_ERROR1;
				}else if(stop == 1){
					soccer_step = STEP_STOP1;
				}else{
					if(mp_Axis.mp_cyclicSetRotary[0].UpdateDone == 1){
						mp_Axis.mp_cyclicSetRotary[0].Update = 0;
						if(mp_Axis.mp_cyclicSetRotary[0].CommandBusy == 0 && mp_Axis.mp_cyclicSetRotary[0].CyclicSetActive == 0){
							soccer_step = STEP_RUN27;
						}
					}
				}
			}
			break;
		case STEP_RUN27:
			{
				mp_Axis.mp_cyclicSetRotary[0].CyclicPosition = 1;
				if(mp_alarmX.mp_core.ActiveAlarms == 1){
					soccer_step = STEP_ERROR1;
				}else if(stop == 1){
					soccer_step = STEP_STOP1;
				}else{
					if(mp_Axis.mp_cyclicSetRotary[0].Info.SlavePosition == -800){
						mp_Axis.mp_cyclicSetRotary[0].CyclicPosition = 0;
						if(mp_Axis.mp_cyclicSetRotary[0].CommandBusy == 0 && mp_Axis.mp_cyclicSetRotary[0].CyclicSetActive == 0){
							soccer_step = STEP_RUN28;
						}
					}
				}
			}
			break;
		case STEP_RUN28:
			{
				mp_Axis.param_cyclicSetRotary[0].Acceleration = 11300;
				mp_Axis.param_cyclicSetRotary[0].Deceleration = 11300;
				mp_Axis.param_cyclicSetRotary[0].PositionModeMaxVelocity = 85000;
				mp_Axis.mp_cyclicSetRotary[0].Velocity 	 = 3000;
				mp_Axis.mp_cyclicSetRotary[0].Position	 = 800;

				mp_Axis.mp_cyclicSetRotary[0].Update = 1;
				if(mp_alarmX.mp_core.ActiveAlarms == 1){
					soccer_step = STEP_ERROR1;
				}else if(stop == 1){
					soccer_step = STEP_STOP1;
				}else{
					if(mp_Axis.mp_cyclicSetRotary[0].UpdateDone == 1){
						mp_Axis.mp_cyclicSetRotary[0].Update = 0;
						if(mp_Axis.mp_cyclicSetRotary[0].CommandBusy == 0 && mp_Axis.mp_cyclicSetRotary[0].CyclicSetActive == 0){
							soccer_step = STEP_RUN29;
						}
					}
				}
			}
			break;
		case STEP_RUN29:
			{
				mp_Axis.mp_cyclicSetRotary[0].CyclicPosition = 1;
				if(mp_alarmX.mp_core.ActiveAlarms == 1){
					soccer_step = STEP_ERROR1;
				}else if(stop == 1){
					soccer_step = STEP_STOP1;
				}else{
					if(mp_Axis.mp_cyclicSetRotary[0].Info.SlavePosition == 800){
						mp_Axis.mp_cyclicSetRotary[0].CyclicPosition = 0;
						if(mp_Axis.mp_cyclicSetRotary[0].CommandBusy == 0 && mp_Axis.mp_cyclicSetRotary[0].CyclicSetActive == 0){
							soccer_step = STEP_RUN30;
						}
					}
				}
			}
			break;
		case STEP_RUN30:
			{
				mp_Axis.param_cyclicSetRotary[0].Acceleration = 1000;
				mp_Axis.param_cyclicSetRotary[0].Deceleration = 1000;
				mp_Axis.param_cyclicSetRotary[0].PositionModeMaxVelocity = 85000;
				mp_Axis.mp_cyclicSetRotary[0].Velocity 	 = 1000;
				mp_Axis.mp_cyclicSetRotary[0].Position	 = 0;

				mp_Axis.mp_cyclicSetRotary[0].Update = 1;
				if(mp_alarmX.mp_core.ActiveAlarms == 1){
					soccer_step = STEP_ERROR1;
				}else if(stop == 1){
					soccer_step = STEP_STOP1;
				}else{
					if(mp_Axis.mp_cyclicSetRotary[0].UpdateDone == 1){
						mp_Axis.mp_cyclicSetRotary[0].Update = 0;
						if(mp_Axis.mp_cyclicSetRotary[0].CommandBusy == 0 && mp_Axis.mp_cyclicSetRotary[0].CyclicSetActive == 0){
							soccer_step = STEP_RUN31;
						}
					}
				}
			}
			break;
		case STEP_RUN31:
			{
				mp_Axis.mp_cyclicSetRotary[0].CyclicPosition = 1;
				if(mp_alarmX.mp_core.ActiveAlarms == 1){
					soccer_step = STEP_ERROR1;
				}else if(stop == 1){
					soccer_step = STEP_STOP1;
				}else{
					if(mp_Axis.mp_cyclicSetRotary[0].Info.SlavePosition == 0){
						mp_Axis.mp_cyclicSetRotary[0].CyclicPosition = 0;
						if(mp_Axis.mp_cyclicSetRotary[0].CommandBusy == 0 && mp_Axis.mp_cyclicSetRotary[0].CyclicSetActive == 0){
							soccer_step = STEP_RUN32; //STEP_RUN8
						}
					}
				}
			}
			break;
		case STEP_RUN32:
			{
				mp_Axis.param_cyclicSetLinear[0].Acceleration = 440000;
				mp_Axis.param_cyclicSetLinear[0].Deceleration = 440000;
				mp_Axis.param_cyclicSetLinear[0].PositionModeMaxVelocity = 30000;
				mp_Axis.mp_cyclicSetLinear[0].Velocity = 20000;
				mp_Axis.mp_cyclicSetLinear[0].Position = 0;

				mp_Axis.mp_cyclicSetLinear[0].Update = 1;
				if(mp_alarmX.mp_core.ActiveAlarms == 1){
					soccer_step = STEP_ERROR1;
				}else if(stop == 1){
					soccer_step = STEP_STOP1;
				}else{
					if(mp_Axis.mp_cyclicSetLinear[0].UpdateDone == 1){
						mp_Axis.mp_cyclicSetLinear[0].Update = 0;
						if(mp_Axis.mp_cyclicSetLinear[0].CommandBusy == 0 && mp_Axis.mp_cyclicSetLinear[0].CyclicSetActive == 0){
							soccer_step = STEP_RUN33;
						}
					}
				}
			}
			break;
		case STEP_RUN33:
			{
				mp_Axis.mp_cyclicSetLinear[0].CyclicPosition = 1;
				if(mp_alarmX.mp_core.ActiveAlarms == 1){
					soccer_step = STEP_ERROR1;
				}else if(stop == 1){
					soccer_step = STEP_STOP1;
				}else{
					if(mp_Axis.mp_cyclicSetLinear[0].Info.SlavePosition == 0){
						mp_Axis.mp_cyclicSetLinear[0].CyclicPosition = 0;
						if(mp_Axis.mp_cyclicSetLinear[0].CommandBusy == 0 && mp_Axis.mp_cyclicSetLinear[0].CyclicSetActive == 0){
							soccer_step = STEP_RUN34;
						}
					}
				}
			}
			break;
		case STEP_RUN34:
			{
				mp_Axis.param_cyclicSetRotary[0].Acceleration = 3900000;
				mp_Axis.param_cyclicSetRotary[0].Deceleration = 3900000;
				mp_Axis.param_cyclicSetRotary[0].PositionModeMaxVelocity = 85000;
				mp_Axis.mp_cyclicSetRotary[0].Velocity 	 = 84000;
				mp_Axis.mp_cyclicSetRotary[0].Position	 = -800;

				mp_Axis.mp_cyclicSetRotary[0].Update = 1;
				if(mp_alarmX.mp_core.ActiveAlarms == 1){
					soccer_step = STEP_ERROR1;
				}else if(stop == 1){
					soccer_step = STEP_STOP1;
				}else{
					if(mp_Axis.mp_cyclicSetRotary[0].UpdateDone == 1){
						mp_Axis.mp_cyclicSetRotary[0].Update = 0;
						if(mp_Axis.mp_cyclicSetRotary[0].CommandBusy == 0 && mp_Axis.mp_cyclicSetRotary[0].CyclicSetActive == 0){
							soccer_step = STEP_RUN35;
						}
					}
				}
			}
			break;
		case STEP_RUN35:
			{
				mp_Axis.mp_cyclicSetRotary[0].CyclicPosition = 1;
				if(mp_alarmX.mp_core.ActiveAlarms == 1){
					soccer_step = STEP_ERROR1;
				}else if(stop == 1){
					soccer_step = STEP_STOP1;
				}else{
					if(mp_Axis.mp_cyclicSetRotary[0].Info.SlavePosition == -800){
						mp_Axis.mp_cyclicSetRotary[0].CyclicPosition = 0;
						if(mp_Axis.mp_cyclicSetRotary[0].CommandBusy == 0 && mp_Axis.mp_cyclicSetRotary[0].CyclicSetActive == 0){
							soccer_step = STEP_RUN36;
						}
					}
				}
			}
			break;
		case STEP_RUN36:
			{
				mp_Axis.param_cyclicSetRotary[0].Acceleration = 3900000;
				mp_Axis.param_cyclicSetRotary[0].Deceleration = 3900000;
				mp_Axis.param_cyclicSetRotary[0].PositionModeMaxVelocity = 85000;
				mp_Axis.mp_cyclicSetRotary[0].Velocity 	 = 84000;
				mp_Axis.mp_cyclicSetRotary[0].Position	 = 800;

				mp_Axis.mp_cyclicSetRotary[0].Update = 1;
				if(mp_alarmX.mp_core.ActiveAlarms == 1){
					soccer_step = STEP_ERROR1;
				}else if(stop == 1){
					soccer_step = STEP_STOP1;
				}else{
					if(mp_Axis.mp_cyclicSetRotary[0].UpdateDone == 1){
						mp_Axis.mp_cyclicSetRotary[0].Update = 0;
						if(mp_Axis.mp_cyclicSetRotary[0].CommandBusy == 0 && mp_Axis.mp_cyclicSetRotary[0].CyclicSetActive == 0){
							soccer_step = STEP_RUN37;
						}
					}
				}
			}
			break;
		case STEP_RUN37:
			{
				mp_Axis.mp_cyclicSetRotary[0].CyclicPosition = 1;
				if(mp_alarmX.mp_core.ActiveAlarms == 1){
					soccer_step = STEP_ERROR1;
				}else if(stop == 1){
					soccer_step = STEP_STOP1;
				}else{
					if(mp_Axis.mp_cyclicSetRotary[0].Info.SlavePosition == 800){
						mp_Axis.mp_cyclicSetRotary[0].CyclicPosition = 0;
						if(mp_Axis.mp_cyclicSetRotary[0].CommandBusy == 0 && mp_Axis.mp_cyclicSetRotary[0].CyclicSetActive == 0){
							soccer_step = STEP_RUN38;
						}
					}
				}
			}
			break;
		case STEP_RUN38:
			{
				mp_Axis.param_cyclicSetRotary[0].Acceleration = 61300;
				mp_Axis.param_cyclicSetRotary[0].Deceleration = 61300;
				mp_Axis.param_cyclicSetRotary[0].PositionModeMaxVelocity = 85000;
				mp_Axis.mp_cyclicSetRotary[0].Velocity 	 = 7000;
				mp_Axis.mp_cyclicSetRotary[0].Position	 = 0;

				mp_Axis.mp_cyclicSetRotary[0].Update = 1;
				if(mp_alarmX.mp_core.ActiveAlarms == 1){
					soccer_step = STEP_ERROR1;
				}else if(stop == 1){
					soccer_step = STEP_STOP1;
				}else{
					if(mp_Axis.mp_cyclicSetRotary[0].UpdateDone == 1){
						mp_Axis.mp_cyclicSetRotary[0].Update = 0;
						if(mp_Axis.mp_cyclicSetRotary[0].CommandBusy == 0 && mp_Axis.mp_cyclicSetRotary[0].CyclicSetActive == 0){
							soccer_step = STEP_RUN39;
						}
					}
				}
			}
			break;
		case STEP_RUN39:
			{
				mp_Axis.mp_cyclicSetRotary[0].CyclicPosition = 1;
				if(mp_alarmX.mp_core.ActiveAlarms == 1){
					soccer_step = STEP_ERROR1;
				}else if(stop == 1){
					soccer_step = STEP_STOP1;
				}else{
					if(mp_Axis.mp_cyclicSetRotary[0].Info.SlavePosition == 0){
						mp_Axis.mp_cyclicSetRotary[0].CyclicPosition = 0;
						if(mp_Axis.mp_cyclicSetRotary[0].CommandBusy == 0 && mp_Axis.mp_cyclicSetRotary[0].CyclicSetActive == 0){
							soccer_step = STEP_RUN8;
						}
					}
				}
			}
			break;
		case STEP_RUN40:
			{
				if(mp_alarmX.mp_core.ActiveAlarms == 1){
					soccer_step = STEP_ERROR1;
				}else if(stop == 1){
					soccer_step = STEP_STOP1;
				}else{
				}
			}
			break;
		case STEP_STOP1:
			{
				start = 0;
				mp_Axis.mp_axisLinear[0].Stop = 1;
				mp_Axis.mp_axisRotary[0].Stop = 1;

				if(mp_alarmX.mp_core.ActiveAlarms == 1){
					soccer_step = STEP_ERROR1;
				}else if(stop == 0){
					mp_Axis.mp_axisLinear[0].Stop = 0;
					mp_Axis.mp_axisRotary[0].Stop = 0;
					soccer_step = STEP_INITIALIZATION0;
				}
			}
			break;
		case STEP_ERROR1:
			{
				start = 0;
				stop  = 0;
				mp_Axis.mp_axisLinear[0].Stop = 0;
				mp_Axis.mp_axisRotary[0].Stop = 0;
				mp_Axis.mp_axisLinear[0].Power = 0;
				mp_Axis.mp_axisRotary[0].Power = 0;

				mp_Axis.mp_axisLinear[0].ErrorReset = 1;
				mp_Axis.mp_axisRotary[0].ErrorReset = 1;

				if(mp_Axis.mp_axisLinear[0].Error == 0 && mp_Axis.mp_axisRotary[0].Error == 0){
					mp_Axis.mp_axisLinear[0].ErrorReset = 0;
					mp_Axis.mp_axisRotary[0].ErrorReset = 0;

					soccer_step = STEP_INITIALIZATION0;
				}

			}
			break;
		case STEP_ERROR2:
			{
				mp_Axis.mp_axisLinear[0].ErrorReset = 1;
				mp_Axis.mp_axisRotary[0].ErrorReset = 1;

				if(mp_Axis.mp_axisLinear[0].StatusID >= 0 && mp_Axis.mp_axisRotary[0].StatusID >= 0){
					mp_Axis.mp_axisLinear[0].ErrorReset = 0;
					mp_Axis.mp_axisRotary[0].ErrorReset = 0;

					soccer_step = STEP_INITIALIZATION0;
				}
			}
			break;
	}

    /************************** Call function & function blocks **************************/
    // AlarmX
    MpAlarmXCore(&mp_alarmX.mp_core);
    MpAlarmXListUI(&mp_alarmX.mp_listUI);
    MpAlarmXHistory(&mp_alarmX.mp_history);
    MpAlarmXHistoryUI(&mp_alarmX.mp_historyUI);
    // Active AxisBasic & AxisCyclicSet -> through the individual functions
    start_axesBasic(max_numberOfFormation,&mp_Axis.mp_axisLinear,&mp_Axis.mp_axisRotary);
    start_axesCyclic(max_numberOfFormation,&mp_Axis.mp_cyclicSetLinear,&mp_Axis.mp_cyclicSetRotary);

}
```

### Program Logical/Real_Game/Technology/cam_sens_sd_s (ANSIC) - Lubo,Radek program for real game.

#### Variables.var
```iecst
VAR
	enable : BOOL;
END_VAR
```

#### main_real.c
```c
/*********************************************************************************************
* B&R Automation - Perfection in Automation (https://www.br-automation.com)
    ******************************************************************************************
    * Program 	    : Bachelor's Thesis
    * Author  	    : Lubomir Bubenik, Radek Otradovský
    * Created 	    : date ...
	* University    : Brno University of Technology(BUT)
	* Faculty       : Faculty of Mechanical Engineering(FME), Faculty of Electrical Engineering and Communication(FEEC)
**********************************************************************************************
* Implementation OF PROGRAM cam_sens_sd_s(Real_Game/Technology/sim_cam_sens_sd_s/main_real.c)
**********************************************************************************************/

#include <bur/plctypes.h>

#ifdef _DEFAULT_INCLUDES
#include <AsDefault.h>
#endif

_GLOBAL FBCamera_typ FBCamera_0;

_GLOBAL Light_typ Light_0;

void _INIT ProgramInit(void)
{
	FBCamera_0.Enable = 0;
}

void _CYCLIC ProgramCyclic(void)
{

	FBCamera(&FBCamera_0);
	Light(&Light_0);

}

void _EXIT ProgramExit(void)
{
	// Insert code here

}
```

### Program Logical/Real_Game/Technology/Lights_control (ANSIC)

#### Main.c - Init, cyclic, exit code
```c
#include <bur/plctypes.h>
#include "Bar_Light.h"

#ifdef _DEFAULT_INCLUDES
	#include <AsDefault.h>
#endif

_GLOBAL Light_typ Light_0;

void _INIT ProgramInit(void)
{
	Light_0.Enable = 1;
	Light(&Light_0);
	Light_0.PowerOn = 1;
}

void _CYCLIC ProgramCyclic(void)
{
	// Lights
	Light(&Light_0);

}
```


- Data object Logical/Real_Game/Motion_Test/Linear/gkLinearWobj/gkLinearWa (Apt) (no source held here)

- Data object Logical/Real_Game/Motion_Test/Linear/gkLinearWobj/gkLinearWi (Ax) (no source held here)

### Package Logical/Real_Game/Motion_Test/Rotary/gkRotaryWobj - gkRotaryWobj

### Data object Logical/Real_Game/Motion_Test/Rotary/gkRotaryWobj/gkRotaryWi (Ax)

#### gkRotaryWi.ax
```
InitParameter (Version=3.14.3, NcSwId=Acp10)
  ACP10AXIS_typ:
    dig_in:
      level:
        reference = ncACTIV_HI
        pos_hw_end = ncACTIV_HI
        neg_hw_end = ncACTIV_HI
        trigger1 = ncACTIV_HI
        trigger2 = ncACTIV_HI
    encoder_if:
      parameter:
        count_dir = ncSTANDARD
        scaling:
          load:
            units = 3600
            rev_motor = 1
    limit:
      parameter:
        v_pos = 100000.0
        v_neg = 100000.0
        a1_pos = 4000000.0
        a2_pos = 4000000.0
        a1_neg = 4000000.0
        a2_neg = 4000000.0
        t_jolt = 0.0
        t_in_pos = 0
        pos_sw_end = 3600
        neg_sw_end = -3600
        ds_warning = 3600.0
        ds_stop = 3600.0
        a_stop = 1.0e30
        dv_stop = 0
        dv_stop_mode = ncOFF
    controller:
      mode = ncPOSITION
      position:
        kv = 350.0
        tn = 0
        t_predict = 0.0004
        t_total = 0.0004
        p_max = 1.0e30
        i_max = 1.0E+30
      speed:
        kv = 2.5
        tn = 0
        t_filter = 0.0
        isq_filter1:
          type = ncOFF
          a0 = 0.0
          a1 = 0.0
          b0 = 0.0
          b1 = 0.0
          b2 = 0.0
          c0_par_id = 0
          c1_par_id = 0
        isq_filter2:
          type = ncOFF
          a0 = 0.0
          a1 = 0.0
          b0 = 0.0
          b1 = 0.0
          b2 = 0.0
          c0_par_id = 0
          c1_par_id = 0
        isq_filter3:
          type = ncOFF
          a0 = 0.0
          a1 = 0.0
          b0 = 0.0
          b1 = 0.0
          b2 = 0.0
          c0_par_id = 0
          c1_par_id = 0
      uf:
        type = ncLINEAR
        auto_config = ncMOTOR_PAR
        u0 = 0
        un = 0
        fn = 50.0
        k_f_slip = 0
      ff:
        torque_load = 0.0
        torque_pos = 0.0
        torque_neg = 0.0
        kv_torque = 0.0120116
        inertia = 0.000109668
        t_filter_a = 0.0
    move:
      stop:
        parameter[0]:
          decel_ramp = ncA_LIMIT
          controller = ncON
        parameter[1]:
          decel_ramp = ncA_LIMIT
          controller = ncON
        parameter[2]:
          decel_ramp = ncA_LIMIT
          controller = ncON
        parameter[3]:
          decel_ramp = ncA_LIMIT
          controller = ncON
        quickstop:
          decel_ramp = ncA_LIMIT
        drive_error:
          decel_ramp = ncA_LIMIT
      homing:
        parameter:
          s = 0
          v_switch = 50.0
          v_trigger = 5.0
          a = 500.0
          mode = ncDIRECT
          edge_sw = ncPOSITIVE
          start_dir = ncPOSITIVE
          trigg_dir = ncPOSITIVE
          ref_pulse = ncOFF
          fix_dir = ncOFF
          tr_s_block = 0
          torque_lim = 0
          ds_block = 0
          ds_stop = 0
      basis:
        parameter:
          v_pos = 84000.0
          v_neg = 84000.0
          a1_pos = 3850000.0
          a2_pos = 3850000.0
          a1_neg = 3850000.0
          a2_neg = 3850000.0
    message:
      text:
        parameter:
          format = ncBREAK
          columns = 80
          data_modul = acp10etxen
```

### Package Logical/Real_Game/Motion_RG/gkRotaryDobj - gkRotaryDobj

### Data object Logical/Real_Game/Motion_RG/gkRotaryDobj/gkRotaryDa (Apt)

#### gkRotaryDa.apt
```
AcoposParameterTable:
  Root Parameters:
    719 = 1 (Name=ENCOD_CMD)  // Encoder1: Encoder command
```

### Data object Logical/Real_Game/Motion_RG/gkRotaryDobj/gkRotaryDi (Ax)

#### gkRotaryDi.ax
```
InitParameter (Version=3.13.1, NcSwId=Acp10)
  ACP10AXIS_typ:
    dig_in:
      level:
        reference = ncACTIV_HI
        pos_hw_end = ncACTIV_HI
        neg_hw_end = ncACTIV_HI
        trigger1 = ncACTIV_HI
        trigger2 = ncACTIV_HI
    encoder_if:
      parameter:
        count_dir = ncSTANDARD
        scaling:
          load:
            units = 3600
            rev_motor = 1
    limit:
      parameter:
        v_pos = 100000.0
        v_neg = 100000.0
        a1_pos = 4000000.0
        a2_pos = 4000000.0
        a1_neg = 4000000.0
        a2_neg = 4000000.0
        t_jolt = 0
        t_in_pos = 0
        pos_sw_end = 3600
        neg_sw_end = -3600
        ds_warning = 3600.0
        ds_stop = 3600.0
        a_stop = 1.0e30
        dv_stop = 0
        dv_stop_mode = ncOFF
    controller:
      mode = ncPOSITION
      position:
        kv = 350.0
        tn = 0
        t_predict = 0.0004
        t_total = 0.0004
        p_max = 1.0e30
        i_max = 1.0E+30
      speed:
        kv = 2.5
        tn = 0
        t_filter = 0.0
        isq_filter1:
          type = ncOFF
          a0 = 0.0
          a1 = 0.0
          b0 = 0.0
          b1 = 0.0
          b2 = 0.0
          c0_par_id = 0
          c1_par_id = 0
        isq_filter2:
          type = ncOFF
          a0 = 0.0
          a1 = 0.0
          b0 = 0.0
          b1 = 0.0
          b2 = 0.0
          c0_par_id = 0
          c1_par_id = 0
        isq_filter3:
          type = ncOFF
          a0 = 0.0
          a1 = 0.0
          b0 = 0.0
          b1 = 0.0
          b2 = 0.0
          c0_par_id = 0
          c1_par_id = 0
      uf:
        type = ncLINEAR
        auto_config = ncMOTOR_PAR
        u0 = 0
        un = 0
        fn = 50.0
        k_f_slip = 0
      ff:
        torque_load = 0.0
        torque_pos = 0.0
        torque_neg = 0.0
        kv_torque = 0.0120116
        inertia = 0.000109668
        t_filter_a = 0.0
    move:
      stop:
        parameter[0]:
          decel_ramp = ncA_LIMIT
          controller = ncON
        parameter[1]:
          decel_ramp = ncA_LIMIT
          controller = ncON
        parameter[2]:
          decel_ramp = ncA_LIMIT
          controller = ncON
        parameter[3]:
          decel_ramp = ncA_LIMIT
          controller = ncON
        quickstop:
          decel_ramp = ncA_LIMIT
        drive_error:
          decel_ramp = ncA_LIMIT
      homing:
        parameter:
          s = 0
          v_switch = 50.0
          v_trigger = 5.0
          a = 500.0
          mode = ncDIRECT
          edge_sw = ncPOSITIVE
          start_dir = ncPOSITIVE
          trigg_dir = ncPOSITIVE
          ref_pulse = ncOFF
          fix_dir = ncOFF
          tr_s_block = 0
          torque_lim = 0
          ds_block = 0
          ds_stop = 0
      basis:
        parameter:
          v_pos = 84000.0
          v_neg = 84000.0
          a1_pos = 3850000.0
          a2_pos = 3850000.0
          a1_neg = 3850000.0
          a2_neg = 3850000.0
    message:
      text:
        parameter:
          format = ncBREAK
          columns = 80
          data_modul = acp10etxen
```


- Data object Logical/Real_Game/Motion_RG/gkRotaryGobj/gkRotaryGa (Apt) (no source held here)

- Data object Logical/Real_Game/Motion_RG/gkRotaryGobj/gkRotaryGi (Ax) (no source held here)

### Package Logical/Real_Game/Motion_RG/gkLinearDobj - gkLinearDobj

- Data object Logical/Real_Game/Motion_RG/gkLinearDobj/gkLinearDa (Apt) (no source held here)

### Data object Logical/Real_Game/Motion_RG/gkLinearDobj/gkLinearDi (Ax)

#### gkLinearDi.ax
```
InitParameter (Version=3.13.1, NcSwId=Acp10)
  ACP10AXIS_typ:
    dig_in:
      level:
        reference = ncACTIV_HI
        pos_hw_end = ncACTIV_HI
        neg_hw_end = ncACTIV_HI
        trigger1 = ncACTIV_HI
        trigger2 = ncACTIV_HI
    encoder_if:
      parameter:
        count_dir = ncSTANDARD
        scaling:
          load:
            units = 200
            rev_motor = 1
    limit:
      parameter:
        v_pos = 30000.0
        v_neg = 30000.0
        a1_pos = 490000.0
        a2_pos = 490000.0
        a1_neg = 490000.0
        a2_neg = 490000.0
        t_jolt = 0
        t_in_pos = 0
        pos_sw_end = 900
        neg_sw_end = -900
        ds_warning = 30.0
        ds_stop = 170.0
        a_stop = 1.0e30
        dv_stop = 0
        dv_stop_mode = ncOFF
    controller:
      mode = ncPOSITION
      position:
        kv = 120.0
        tn = 0
        t_predict = 0.0004
        t_total = 0.0004
        p_max = 1.0e30
        i_max = 1.0E+30
      speed:
        kv = 0.25
        tn = 0
        t_filter = 0.01
        isq_filter1:
          type = ncNOTCH
          a0 = 2299.41
          a1 = 400.0
          b0 = 0.0
          b1 = 0.0
          b2 = 0.0
          c0_par_id = 0
          c1_par_id = 0
        isq_filter2:
          type = ncOFF
          a0 = 0.0
          a1 = 0.0
          b0 = 0.0
          b1 = 0.0
          b2 = 0.0
          c0_par_id = 0
          c1_par_id = 0
        isq_filter3:
          type = ncOFF
          a0 = 0.0
          a1 = 0.0
          b0 = 0.0
          b1 = 0.0
          b2 = 0.0
          c0_par_id = 0
          c1_par_id = 0
      uf:
        type = ncLINEAR
        auto_config = ncMOTOR_PAR
        u0 = 0
        un = 0
        fn = 50.0
        k_f_slip = 0
      ff:
        torque_load = 0.0
        torque_pos = 0.00691027
        torque_neg = 0.00674195
        kv_torque = 0.000864945
        inertia = 1.13117E-05
        t_filter_a = 0.0
    move:
      stop:
        parameter[0]:
          decel_ramp = ncA_LIMIT
          controller = ncON
        parameter[1]:
          decel_ramp = ncA_LIMIT
          controller = ncON
        parameter[2]:
          decel_ramp = ncA_LIMIT
          controller = ncON
        parameter[3]:
          decel_ramp = ncA_LIMIT
          controller = ncON
        quickstop:
          decel_ramp = ncA_LIMIT
        drive_error:
          decel_ramp = ncA_LIMIT
      homing:
        parameter:
          s = 900
          v_switch = 350.0
          v_trigger = 350.0
          a = 4000.0
          mode = ncBLOCK_TORQUE
          edge_sw = ncPOSITIVE
          start_dir = ncPOSITIVE
          trigg_dir = ncNEGATIVE
          ref_pulse = ncOFF
          fix_dir = ncOFF
          tr_s_block = 0
          torque_lim = 0.02
          ds_block = 0.0
          ds_stop = 1000.0
      basis:
        parameter:
          v_pos = 20000.0
          v_neg = 20000.0
          a1_pos = 400000.0
          a2_pos = 400000.0
          a1_neg = 400000.0
          a2_neg = 400000.0
    message:
      text:
        parameter:
          format = ncBREAK
          columns = 80
          data_modul = acp10etxen
```

### Package Logical/Real_Game/Motion_RG/gkLinearGobj - gkLinearGobj

- Data object Logical/Real_Game/Motion_RG/gkLinearGobj/gkLinearGa (Apt) (no source held here)

### Data object Logical/Real_Game/Motion_RG/gkLinearGobj/gkLinearGi (Ax)

#### gkLinearGi.ax
```
InitParameter (Version=3.16.2, NcSwId=Acp10)
  ACP10AXIS_typ:
    dig_in:
      level:
        reference = ncACTIV_HI
        pos_hw_end = ncACTIV_HI
        neg_hw_end = ncACTIV_HI
        trigger1 = ncACTIV_HI
        trigger2 = ncACTIV_HI
    encoder_if:
      parameter:
        count_dir = ncSTANDARD
        scaling:
          load:
            units = 1000
            rev_motor = 1
    limit:
      parameter:
        v_pos = 10000
        v_neg = 10000
        a1_pos = 50000
        a2_pos = 50000
        a1_neg = 50000
        a2_neg = 50000
        t_jolt = 0
        t_in_pos = 0
        pos_sw_end = 2000000000
        neg_sw_end = -2000000000
        ds_warning = 500
        ds_stop = 1000
        a_stop = 1.0e30
        dv_stop = 0
        dv_stop_mode = ncOFF
    controller:
      mode = ncPOSITION
      position:
        kv = 50
        tn = 0
        t_predict = 0.0004
        t_total = 0.0004
        p_max = 1.0e30
        i_max = 0
      speed:
        kv = 2.0
        tn = 0
        t_filter = 0.0
        isq_filter1:
          type = ncOFF
          a0 = 0.0
          a1 = 0.0
          b0 = 0.0
          b1 = 0.0
          b2 = 0.0
          c0_par_id = 0
          c1_par_id = 0
        isq_filter2:
          type = ncOFF
          a0 = 0.0
          a1 = 0.0
          b0 = 0.0
          b1 = 0.0
          b2 = 0.0
          c0_par_id = 0
          c1_par_id = 0
        isq_filter3:
          type = ncOFF
          a0 = 0.0
          a1 = 0.0
          b0 = 0.0
          b1 = 0.0
          b2 = 0.0
          c0_par_id = 0
          c1_par_id = 0
      uf:
        type = ncLINEAR
        auto_config = ncMOTOR_PAR
        u0 = 0
        un = 0
        fn = 50.0
        k_f_slip = 0
      ff:
        torque_load = 0.0
        torque_pos = 0.0
        torque_neg = 0.0
        kv_torque = 0.0
        inertia = 0.0
        t_filter_a = 0.0
    move:
      stop:
        parameter[0]:
          decel_ramp = ncA_LIMIT
          controller = ncON
        parameter[1]:
          decel_ramp = ncA_LIMIT
          controller = ncON
        parameter[2]:
          decel_ramp = ncA_LIMIT
          controller = ncON
        parameter[3]:
          decel_ramp = ncA_LIMIT
          controller = ncON
        quickstop:
          decel_ramp = ncA_LIMIT
        drive_error:
          decel_ramp = ncA_LIMIT
      homing:
        parameter:
          s = 0
          v_switch = 5000
          v_trigger = 500
          a = 50000
          mode = ncDIRECT
          edge_sw = ncPOSITIVE
          start_dir = ncPOSITIVE
          trigg_dir = ncPOSITIVE
          ref_pulse = ncOFF
          fix_dir = ncOFF
          tr_s_block = 0
          torque_lim = 0
          ds_block = 0
          ds_stop = 0
      basis:
        parameter:
          v_pos = 5000
          v_neg = 5000
          a1_pos = 50000
          a2_pos = 50000
          a1_neg = 50000
          a2_neg = 50000
    message:
      text:
        parameter:
          format = ncBREAK
          columns = 80
          data_modul = acp10etxen
```


- Data object Logical/Real_Game/Motion_RG/gkRotaryFobj/gkRotaryFa (Apt) (no source held here)

- Data object Logical/Real_Game/Motion_RG/gkRotaryFobj/gkRotaryFi (Ax) (no source held here)

- Data object Logical/Real_Game/Motion_RG/gkRotaryMobj/gkRotaryMa (Apt) (no source held here)

- Data object Logical/Real_Game/Motion_RG/gkRotaryMobj/gkRotaryMi (Ax) (no source held here)

- Data object Logical/Real_Game/Motion_RG/gkLinearFobj/gkLinearFa (Apt) (no source held here)

- Data object Logical/Real_Game/Motion_RG/gkLinearFobj/gkLinearFi (Ax) (no source held here)

### Package Logical/Real_Game/Motion_RG/gkLinearMobj - gkLinearMobj

### Data object Logical/Real_Game/Motion_RG/gkLinearMobj/gkLinearMa (Apt)

#### gkLinearMa.apt
```
AcoposParameterTable:
  Root Parameters:
    linMot.xml:
      linMot__PS01-23x80/150x210.xml:
        LinMot: PS01-23x80/150x210  // Version: 1.1
          Motor (Disabled=FALSE)
            30 = 0x0002 (Name=MOTOR_TYPE, Disabled=FALSE)  // Motor: Type
            31 = 0x0203 (Name=MOTOR_COMPATIBILITY, Disabled=FALSE)  // Motor: Software compatibility
            46 = 1 (Name=MOTOR_WIND_CONNECT, Disabled=FALSE)  // Motor: Winding connection
            47 = 1 (Name=MOTOR_POLEPAIRS, Disabled=FALSE)  // Motor: Number of pole-pairs
            1208 = 2 (Name=MOTOR_NUM_PHASES)  // Motor: Number of motor phases
            48 = 72 (Name=MOTOR_VOLTAGE_RATED, Unit=V, Disabled=FALSE)  // Motor: Rated voltage
            49 = 5.209 (Name=MOTOR_VOLTAGE_CONST, Unit=mV*min, Disabled=FALSE)  // Motor: Voltage constant
            51 = 18000 (Name=MOTOR_SPEED_MAX, Unit=1/min, Disabled=FALSE)  // Motor: Maximum speed
            54 = 0.14 (Name=MOTOR_TORQ_MAX, Unit=Nm, Disabled=FALSE)  // Motor: Peak torque
            55 = 0.035 (Name=MOTOR_TORQ_CONST, Unit=Nm/A, Disabled=FALSE)  // Motor: Torque constant
            58 = 4 (Name=MOTOR_CURR_MAX, Unit=A, Disabled=FALSE)  // Motor: Peak current
            60 = 12.5 (Name=MOTOR_STATOR_RESISTANCE, Unit=Ohm, Disabled=FALSE)  // Motor: Stator resistance
            61 = 0.0014 (Name=MOTOR_STATOR_INDUCTANCE, Unit=Henry, Disabled=FALSE)  // Motor: Stator inductance
            62 = 0.0000027 (Name=MOTOR_INERTIA, Unit=kgmp, Disabled=FALSE)  // Motor: Moment of inertia
            63 = 1.5707963 (Name=MOTOR_COMMUT_OFFSET, Unit=rad, Disabled=FALSE)  // Motor: Commutation offset
            276 = 4 (Name=PHASING_MODE, Disabled=FALSE)  // Motor: Phasing: Mode
          50 = 18000 (Name=MOTOR_SPEED_RATED, Unit=1/min, Disabled=FALSE)  // Motor: Rated speed
          Temperature model (Disabled=FALSE)
            56 = 0.82 (Name=MOTOR_CURR_STALL, Unit=A, Disabled=FALSE)  // Motor: Stall current
            57 = 0.82 (Name=MOTOR_CURR_RATED, Unit=A, Disabled=FALSE)  // Motor: Rated current
            52 = 0.03 (Name=MOTOR_TORQ_STALL, Unit=Nm, Disabled=FALSE)  // Motor: Stall torque
            53 = 0.03 (Name=MOTOR_TORQ_RATED, Unit=Nm, Disabled=FALSE)  // Motor: Rated torque
            59 = 0.11 (Name=MOTOR_WIND_CROSS_SECT, Unit=mmp, Disabled=FALSE)  // Motor: Line cross section
            849 = 135.72 (Name=MOTOR_TAU_THERM, Unit=s, Disabled=FALSE)  // Motor: Thermal time constant
            74 = 110 (Name=MOTOR_WIND_TEMP_MAX, Unit=°C, Disabled=FALSE)  // Motor: Limit temperature
            1210 = 2 (Name=MOTOR_TEMPMODEL_REFSENS, Disabled=FALSE)  // Motor: Temperature model: Reference sensor: Parameter-ID
            1211 = 0.2775 (Name=MOTOR_TEMPMODEL_RES1, Unit=K/W, Disabled=FALSE)  // Motor: Temperature model: Thermal resistance 1
            1212 = 17.226 (Name=MOTOR_TEMPMODEL_CAP1, Unit=Ws/K, Disabled=FALSE)  // Motor: Temperature model: Thermal capacity 1
            1213 = 0.4163 (Name=MOTOR_TEMPMODEL_RES2, Unit=K/W, Disabled=FALSE)  // Motor: Temperature model: Thermal resistance 2
            1214 = 0.348 (Name=MOTOR_TEMPMODEL_CAP2, Unit=Ws/K, Disabled=FALSE)  // Motor: Temperature model: Thermal capacity 2
            373 = 4 (Name=TEMP_MOTOR_MODEL_MODE, Disabled=FALSE)  // Motor: Temperature model: Mode
          Brake (Disabled=FALSE)
            42 = 0 (Name=MOTOR_BRAKE_CURR_RATED, Unit=A, Disabled=FALSE)  // Motor holding brake: Rated current
            43 = 0 (Name=MOTOR_BRAKE_TORQ_RATED, Unit=Nm, Disabled=FALSE)  // Motor holding brake: Rated torque
            44 = 0 (Name=MOTOR_BRAKE_ON_TIME, Unit=s, Disabled=FALSE)  // Motor holding brake: Engaging delay
            45 = 0 (Name=MOTOR_BRAKE_OFF_TIME, Unit=s, Disabled=FALSE)  // Motor holding brake: Release delay
          Temperature sensor (Disabled=FALSE)
            64 = 0 (Name=MOTOR_TEMPSENS_PAR1, Disabled=FALSE)  // Temperature sensor: Parameter 1
            65 = 0 (Name=MOTOR_TEMPSENS_PAR2, Disabled=FALSE)  // Temperature sensor: Parameter 2
            66 = 0 (Name=MOTOR_TEMPSENS_PAR3, Disabled=FALSE)  // Temperature sensor: Parameter 3
            67 = 0 (Name=MOTOR_TEMPSENS_PAR4, Disabled=FALSE)  // Temperature sensor: Parameter 4
            68 = 0 (Name=MOTOR_TEMPSENS_PAR5, Disabled=FALSE)  // Temperature sensor: Parameter 5
            69 = 0 (Name=MOTOR_TEMPSENS_PAR6, Disabled=FALSE)  // Temperature sensor: Parameter 6
            70 = 0 (Name=MOTOR_TEMPSENS_PAR7, Disabled=FALSE)  // Temperature sensor: Parameter 7
            71 = 0 (Name=MOTOR_TEMPSENS_PAR8, Disabled=FALSE)  // Temperature sensor: Parameter 8
            72 = 0 (Name=MOTOR_TEMPSENS_PAR9, Disabled=FALSE)  // Temperature sensor: Parameter 9
            73 = 0 (Name=MOTOR_TEMPSENS_PAR10, Disabled=FALSE)  // Temperature sensor: Parameter 10
          Encoder:
            652 = 0 (Name=MOTOR_ENCOD_ATTR, Disabled=FALSE)  // Motor: Encoder: Attribute
            1209 = 110 (Name=MOTOR_ENCOD_TEMP_LIM, Unit=°C, Disabled=FALSE)  // Motor: Encoder: Limit Temperature
            97 = ncLINMOT (Name=ENCOD_TYPE)  // Encoder1: Type
            109 = 16384 (Name=SCALE_ENCOD_INCR)  // Encoder1: Encoder scaling: increments per SCALE_ENCOD_MOTOR_REV motor revolutions
```

### Data object Logical/Real_Game/Motion_RG/gkLinearMobj/gkLinearMi (Ax)

- Visualisation Logical/mappView (not shown)

- Project.language (not shown)

### Program Logical/Program (ANSIC)

#### Main.c - Init, cyclic, exit code
```c
#include <bur/plctypes.h>
#include <AsIecCon.h>
#include <sys_lib.h>

#ifdef _DEFAULT_INCLUDES
	#include <AsDefault.h>
#endif

_GLOBAL FBCamera_typ FBCamera_0;

void _INIT ProgramInit(void)
{
	FBCamera_0.Enable = 0;
}

void _CYCLIC ProgramCyclic(void)
{
	FBCamera(&FBCamera_0);

}

void _EXIT ProgramExit(void)
{
	// Insert code here

}
```

Listed in the project but not available here: Logical/Global.typ, Logical/Libraries/rp_library/rp_funcx1/start_virtualAxis.c, Logical/Libraries/RO_LB_ScoreDetection/Scorkeeper/Types.typ, Logical/Libraries/RO_LB_ScoreDetection/Scorkeeper/Constants.var, Logical/Libraries/RO_LB_ScoreDetection/Scorkeeper/Scorkeeper.fun, Logical/Libraries/RO_Sensors/Library/Constants.var, Logical/Libraries/RO_Sensors/Library/Variables.var, Logical/Libraries/RO_Sensors/ro_sensors/Constants.var, Logical/Libraries/LB_Camera/Camera/Camera.fun, Logical/Libraries/LB_Camera/Bar_Light/Types.typ, Logical/Libraries/LB_Camera/Bar_Light/Constants.var, Logical/Libraries/LB_Camera/Bar_Light/Bar_Light.fun, Logical/Simulation/Technology/sim_cam_sens_sd_s/Types.typ, Logical/Simulation/Technology/sim_cam_sens_sd_s/Variables.var, Logical/Real_Game/Technology/Lights_control/Types.typ, Logical/Real_Game/Technology/Lights_control/Variables.var, Logical/Connection, Logical/Program/Types.typ, Logical/Program/Variables.var
